FUNCTION_BLOCK FB_HMI_CO2_PRESSURE_CONTROL EXTENDS FB_HMI_COMPONENT
VAR_INPUT
END_VAR
VAR_OUTPUT
END_VAR
VAR
END_VAR
VAR_IN_OUT
	{attribute 'OPC.UA.DA' := '0'}
	fbInstance		: FB_NOTT_CO2_PRESSURE_CONTROL;


END_VAR


fbHealthStatus( 
				bIsEnabled:= TRUE, 
				bIsGood := NOT fbInstance.stat.bError,
				bHasWarning := fbInstance.stat.bWarning
				);
				
fbBusyStatus(
				bIsBusy := fbInstance.stat.bBusy,
				bIsEnabled := TRUE);
				
M_UpdateStatusColor();

END_FUNCTION_BLOCK

(* stored: Version 1.1.0.1, ProductVersion 3.1.4024.14
   POU FB_HMI_CO2_PRESSURE_CONTROL: Id {955e6e71-98f5-45d7-bed8-b93f36300160}, SpecialFunc None *)
